# B&R Automation Studio project BaseProject (part 6)

#### Main.st
```iecst
(*******************************************************************************
 * Copyright: B&R Industrial Automation
 * Author:    Tyler Matijevich
 * Created:   November 5, 2020/12:35
********************************************************************************
 * Description: Control program to handle assembly power commands and error
 statuses
********************************************************************************)

PROGRAM _INIT

END_PROGRAM

PROGRAM _CYCLIC

	fbTrakModule(MpLink := ADR(TrackInterface.ModulePml),
					Enable := TRUE,
					Parameters := ADR(parTrakModule));

	// Reset command if no error
	IF gTrakSystem.Asm.Status.Error = FALSE THEN
		gTrakSystem.Asm.Cmd.ErrorReset := FALSE; // Force this command to reset
	END_IF

	(****************************************************************************************************
	****************************************************************************************************)
	(*
		Interrupts:
		1. Error status
		2. Stop command
		3. Read error
		4. ErrorStop state
	*)

	// 1. Skip remaining interrupt checks when an error exists
	IF gTrakSystem.Asm.Status.Error OR ShInit.Status.Error THEN
		// Go to ERROR
		AssemblyState := ASM_STATE_ERROR;

	// 2. Accept stop command
	ELSIF gTrakSystem.Asm.Cmd.Stop THEN
		// Power off if powering or powered on
		IF gTrakSystem.Asm.Status.Homing OR gTrakSystem.Asm.Status.Ready THEN
			// Execute the power off command. Execute should not be true in either of these states
			fbAsmPowerOff.Execute := TRUE;
		END_IF

		// Go to OFF
		AssemblyState := ASM_STATE_OFF;

	// 3. The assembly read function blocks are in error
	ELSIF fbAsmReadStatus.Error OR fbAsmReadInfo.Error THEN
		// Log event
		// Set error status and go to ERROR
		gTrakSystem.Asm.Status.Error	:= TRUE;
		AssemblyState 				:= ASM_STATE_ERROR;

	// 4. Assembly in ErrorStop
	ELSIF gTrakSystem.Asm.Status.ErrorStop AND fbAsmReset.Busy = FALSE THEN
		// Log event
		// Set error status and go to ERROR
		gTrakSystem.Asm.Status.Error	:= TRUE;
		AssemblyState 				:= ASM_STATE_ERROR;

	END_IF

	(****************************************************************************************************
	****************************************************************************************************)
	// Main assembly state machine
	CASE AssemblyState OF
		// ----------------------------------------------------------------------------------------------------
		// OFF
		ASM_STATE_OFF:
			// Accept AsmPowerOff command
			IF fbAsmPowerOff.Done THEN
				// Reset execution
				fbAsmPowerOff.Execute := FALSE;

			ELSIF fbAsmPowerOff.Error THEN
				// Log event
				// Set error status and go to ERROR
				gTrakSystem.Asm.Status.Error	:= TRUE;
				AssemblyState 				:= ASM_STATE_ERROR;

			// Accept AsmReset command
			ELSIF fbAsmReset.Done THEN
				// Reset execution
				fbAsmReset.Execute := FALSE;

			ELSIF fbAsmReset.Error THEN
				// Log event
				// Set error status and go to ERROR
				gTrakSystem.Asm.Status.Error	:= TRUE;
				AssemblyState 				:= ASM_STATE_ERROR;

			// Wait for power command and assembly conditions
			ELSIF gTrakSystem.Asm.Cmd.Power AND gTrakSystem.Asm.Cmd.Stop = FALSE // Read input commands
			  AND gTrakSystem.Asm.Status.Disabled AND gTrakSystem.Asm.Status.ReadyForPowerOn // Check assembly statuses
			  AND fbAsmPowerOff.Execute = FALSE AND fbAsmReset.Execute = FALSE
			  AND MpPackMLStateIsActive(TrackInterface.ModulePml,mpPACKML_STATE_EXECUTE,1)
			  	THEN // Check other function block execution
				// Power on the assembly
				fbAsmPowerOn.Execute := TRUE;

				// Go to POWER
				AssemblyState := ASM_STATE_POWER;

			END_IF

		// ----------------------------------------------------------------------------------------------------
		// POWER
		ASM_STATE_POWER:
			// Wait for the power on command to complete, ensure correct statuses
			IF fbAsmPowerOn.Done AND gTrakSystem.Asm.Status.Ready AND gTrakSystem.Asm.Status.PowerOn THEN
				// Reset execution
				fbAsmPowerOn.Execute := FALSE;

				// Go to READY
				AssemblyState := ASM_STATE_READY;

//				// Check shuttle initialization for ready status
//				IF ShInit.Status.Ready THEN
//					// Start the shuttle initialization
//					ShInit.Cmd.Start := TRUE;
//
//					// Go to INIT
//					AssemblyState := ASM_STATE_INIT;
//
//				ELSE
//					// Log event
//					// Set error status and go to ERROR
//					gTrakSystem.Asm.Status.Error	:= TRUE;
//					AssemblyState 				:= ASM_STATE_ERROR;
//
//				END_IF

			ELSIF fbAsmPowerOn.Error THEN
				// Log event
				// Set error status and go to ERROR
				gTrakSystem.Asm.Status.Error	:= TRUE;
				AssemblyState 				:= ASM_STATE_ERROR;

			// Check if the assembly suddenly loses power
			ELSIF (gTrakSystem.Asm.Status.Disabled OR gTrakSystem.Asm.Status.PowerOn = FALSE)
			  AND fbAsmPowerOn.Execute = FALSE THEN
				// Log event
				// Set error status and go to ERROR
				gTrakSystem.Asm.Status.Error	:= TRUE;
				AssemblyState 				:= ASM_STATE_ERROR;

			END_IF

		// ----------------------------------------------------------------------------------------------------
		// INIT
		ASM_STATE_INIT:
		// Go to READY
				AssemblyState := ASM_STATE_READY;

			// Wait for the shuttle initialization to complete
//			IF ShInit.Status.Complete THEN
//				// Reset command
//				ShInit.Cmd.Start := FALSE;
//
//				// Go to READY
//				AssemblyState := ASM_STATE_READY;
//
//			ELSIF ShInit.Status.Error THEN
//				// Log event
//				// Set error status and go to ERROR
//				gTrakSystem.Asm.Status.Error	:= TRUE;
//				AssemblyState 				:= ASM_STATE_ERROR;
//
//			END_IF

		// ----------------------------------------------------------------------------------------------------
		// READY
		ASM_STATE_READY:
			// Check if the assembly suddenly becomes disabled
			IF gTrakSystem.Asm.Status.Disabled THEN
				// Log event
				// Set error status and go to ERROR
				gTrakSystem.Asm.Status.Error	:= TRUE;
				AssemblyState 				:= ASM_STATE_ERROR;

			END_IF

		// ----------------------------------------------------------------------------------------------------
		// ERROR
		ASM_STATE_ERROR:
			// Wait for an error reset command
			IF gTrakSystem.Asm.Cmd.ErrorReset THEN
				// If ErrorStop, reset the assembly
				IF gTrakSystem.Asm.Status.ErrorStop AND fbAsmReset.Error = FALSE THEN
					// Execute an assembly reset
					fbAsmReset.Execute := TRUE;

					// Reset other function block's execution
					fbAsmPowerOn.Execute 	:= FALSE;
					fbAsmPowerOff.Execute	:= FALSE;

				// If powered
				ELSIF (gTrakSystem.Asm.Status.Homing OR gTrakSystem.Asm.Status.Ready) AND fbAsmPowerOff.Error = FALSE THEN
					// Power off the assembly
					fbAsmPowerOff.Execute := TRUE;

					// Reset other function block's execution
					fbAsmPowerOn.Execute 	:= FALSE;
					fbAsmReset.Execute		:= FALSE;

				ELSE
					// Reset all function block's execution
					fbAsmPowerOn.Execute 	:= FALSE;
					fbAsmPowerOff.Execute	:= FALSE;
					fbAsmReset.Execute		:= FALSE;

				END_IF // Check assembly state

				// Reset the error bit and go back to OFF
				gTrakSystem.Asm.Status.Error	:= FALSE;
				AssemblyState				:= ASM_STATE_OFF;

			END_IF

	END_CASE // Assembly state machine

	// Call all mapp Trak function blocks
	fbAsmReadStatus(Assembly := ADR(TrackInterface.SampleTrak), Enable := TRUE); // Always enable to reduce logger entries
	fbAsmReadInfo(Assembly := ADR(TrackInterface.SampleTrak), Enable := TRUE); // Always enable to reduce logger entries
	fbAsmPowerOn(Assembly := ADR(TrackInterface.SampleTrak));
	fbAsmPowerOff(Assembly := ADR(TrackInterface.SampleTrak));
	fbAsmReset(Assembly := ADR(TrackInterface.SampleTrak));

	// Update the global status information
	gTrakSystem.Asm.Status.Disabled					:= fbAsmReadStatus.Valid AND fbAsmReadStatus.AssemblyDisabled;
	gTrakSystem.Asm.Status.Homing					:= fbAsmReadStatus.Valid AND fbAsmReadStatus.AssemblyHoming;
	gTrakSystem.Asm.Status.Ready					:= fbAsmReadStatus.Valid AND fbAsmReadStatus.AssemblyReady;
	gTrakSystem.Asm.Status.Stopping					:= fbAsmReadStatus.Valid AND fbAsmReadStatus.AssemblyStopping;
	gTrakSystem.Asm.Status.ErrorStop				:= fbAsmReadStatus.Valid AND fbAsmReadStatus.AssemblyErrorStop;
	gTrakSystem.Asm.Status.CommunicationReady		:= fbAsmReadInfo.Valid AND fbAsmReadInfo.AssemblyInfo.CommunicationReady;
	gTrakSystem.Asm.Status.ReadyForPowerOn			:= fbAsmReadInfo.Valid AND fbAsmReadInfo.AssemblyInfo.ReadyForPowerOn;
	gTrakSystem.Asm.Status.PowerOn					:= fbAsmReadInfo.Valid AND fbAsmReadInfo.AssemblyInfo.PowerOn;
	gTrakSystem.Asm.Status.ShuttlesInErrorStopCount	:= fbAsmReadInfo.AssemblyInfo.ShuttlesInErrorStopCount; // If not valid, assuming these are zero
	gTrakSystem.Asm.Status.StartupCount				:= fbAsmReadInfo.AssemblyInfo.StartupCount;

	// Call all subroutine actions
	ShInit.Cmd.Stop := gTrakSystem.Asm.Status.Ready = FALSE;
//	ShuttleInitialization;

END_PROGRAM

PROGRAM _EXIT

END_PROGRAM
```

### SM11.var
```iecst
(*Shuttle initialization variables*)
VAR
	BufferReturnIndex : TrBaseErrorCodeEnum;
	fbAsmGetShuttle : MC_BR_AsmGetShuttle_AcpTrak;
	fbShCopyUserData : MC_BR_ShCopyUserData_AcpTrak;
END_VAR
```

### Program Logical/Source/SampleTrak/Assembly/SubModule1/ShuttleInit (IEC)

#### Main.st
```iecst
PROGRAM _INIT
	(* Insert code here *)
	 TrakInterface;
END_PROGRAM

PROGRAM _CYCLIC
	// Reset status variables, they will be set in the respective state
	ShInit.Status.Ready 	:= FALSE;
	ShInit.Status.Complete	:= FALSE;

	(*
		Interrupts:
		1. Error status
		2. Stop command
	*)
	// 1. Check error status
	IF ShInit.Status.Error THEN
		// Go to ERROR, skip remaining interrupts
		ShInitState := 255;

	// 2. Accept stop commands
	ELSIF ShInit.Cmd.Stop THEN
		// Reset FB execution
		fbAsmGetShuttle.Enable		:= FALSE;
		fbShCopyUserData.Execute 	:= FALSE;

		// Go to INIT
		ShInitState := 0;

	END_IF

	// Shuttle initialization main state machine
	CASE ShInitState OF
		// ----------------------------------------------------------------------------------------------------
		// INIT
		0:
			// Set the status
			ShInit.Status.Ready := TRUE;

			// Wait to start
			IF ShInit.Cmd.Start AND ShInit.Cmd.Stop = FALSE THEN
				// Clear the shuttle buffer
				BufferReturnIndex := TrBaseClearShBuffer(ADR(gTrakSystem.Buffer), SIZEOF(gTrakSystem.Buffer));
				IF BufferReturnIndex = trBASE_NO_ERROR THEN
					// Enable the assembly get shuttle function block
					fbAsmGetShuttle.Assembly 	:= ADR(TrakInterface.SampleTrak);
					fbAsmGetShuttle.Enable 		:= TRUE;

					// Go to READ
					ShInitState := 10;

				ELSE
					// Log event
					// Set error status and go to ERROR
					ShInit.Status.Error := TRUE;
					ShInitState 		:= 255;

				END_IF
			END_IF // Start

		// ----------------------------------------------------------------------------------------------------
		// READ
		10:
			// Wait for a valid read, then read the shuttle
			IF fbAsmGetShuttle.Valid AND fbAsmGetShuttle.TotalCount > 0 THEN
				// Add the shuttle to the buffer
				BufferReturnIndex := TrBaseAddShToBuffer(fbAsmGetShuttle.Axis, ADR(gTrakSystem.Buffer), SIZEOF(gTrakSystem.Buffer));
				IF BufferReturnIndex = trBASE_NO_ERROR THEN
					// Shuttle added successfully, read the shuttle user data
					fbShCopyUserData.Axis 			:= ADR(fbAsmGetShuttle.Axis);
					fbShCopyUserData.DataAddress	:= ADR(ShuttleUserData);
					fbShCopyUserData.DataSize		:= SIZEOF(ShuttleUserData);
					fbShCopyUserData.Mode			:= mcACPTRAK_USERDATA_GET;
					fbShCopyUserData.Execute		:= TRUE;

					// Go to DATA
					ShInitState := 20;

				ELSE
					// Log event
					// Set error status and go to ERROR
					ShInit.Status.Error := TRUE;
					ShInitState 		:= 255;

				END_IF

			ELSIF fbAsmGetShuttle.Valid AND fbAsmGetShuttle.TotalCount = 0 THEN // No shuttles on the assembly
				// Go straight to the complete state
				ShInitState := 60;

			ELSIF fbAsmGetShuttle.Error THEN
				// Log event
				// Set error status and go to ERROR
				ShInit.Status.Error := TRUE;
				ShInitState 		:= 255;

			END_IF

		// ----------------------------------------------------------------------------------------------------
		// DATA
		20:
			IF fbShCopyUserData.Done THEN
				// Reset the command
				fbShCopyUserData.Execute := FALSE;

				// Go to WRITE
				ShInitState := 30;

			ELSIF fbShCopyUserData.Error THEN
				// Log event
				// Set error status and go to ERROR
				ShInit.Status.Error := TRUE;
				ShInitState 		:= 255;

			END_IF

		// ----------------------------------------------------------------------------------------------------
		// WRITE
		30:
			IF fbShCopyUserData.Done THEN
				// Shuttle user data write complete, shuttle ID set, reset the execution
				fbShCopyUserData.Execute := FALSE;

				// Reset the assembly get shuttle next command
				fbAsmGetShuttle.Next := FALSE;

				// Go to UPDATE
				ShInitState := 40;

			ELSIF fbShCopyUserData.Error THEN
				// Log event
				// Set error status and go to ERROR
				ShInit.Status.Error := TRUE;
				ShInitState 		:= 255;

			ELSE
				// Execute the write command
				fbShCopyUserData.Mode		:= mcACPTRAK_USERDATA_SET;
				fbShCopyUserData.Execute 	:= TRUE;

				// Set the shuttle ID (if not already set)
				ShuttleUserData.ID := fbAsmGetShuttle.AdditionalInfo.ShuttleID;

			END_IF

		// ----------------------------------------------------------------------------------------------------
		// UPDATE
		40:
			// Check for the next shuttle
			IF fbAsmGetShuttle.Valid AND fbAsmGetShuttle.RemainingCount > 0 THEN
				// Issue next command and go back to the READ state
				fbAsmGetShuttle.Next 	:= TRUE;
				ShInitState				:= 10;

			// Check when no shuttles remain
			ELSIF fbAsmGetShuttle.Valid AND fbAsmGetShuttle.RemainingCount = 0 THEN
				// All shuttles have been captured, reset the FB
				fbAsmGetShuttle.Enable := FALSE;

				// Go to DELETE
				ShInitState := 50;

			ELSIF fbAsmGetShuttle.Error THEN
				// Log event
				// Set error status and go to ERROR
				ShInit.Status.Error := TRUE;
				ShInitState 		:= 255;

			END_IF

		// ----------------------------------------------------------------------------------------------------
		// DELETE
		50:
			// Shuttle detection complete, now delete marked shuttles
			gTrakSystem.Tracking.Cmd.Delete := gTrakSystem.Tracking.Status.ShuttlesToBeDeletedCount <> 0;

			// Leave when no shuttles need to be deleted
			IF gTrakSystem.Tracking.Status.ShuttlesToBeDeletedCount = 0 THEN
				// Go to COMPLETE
				ShInitState := 60;
			END_IF

		// ----------------------------------------------------------------------------------------------------
		// COMPLETE
		60:
			// Set the status
			ShInit.Status.Complete := TRUE;

			// Return to INIT when the state command is reset
			IF ShInit.Cmd.Start = FALSE THEN
				// Go to INIT
				ShInitState := 0;
			END_IF

		// ----------------------------------------------------------------------------------------------------
		// ERROR
		255:
			// Wait for error reset command
			IF ShInit.Cmd.ErrorReset THEN
				// Reset the function blocks
				fbAsmGetShuttle.Enable 		:= FALSE;
				fbShCopyUserData.Execute 	:= FALSE;

				// Reset the error bit and go to INIT
				ShInit.Status.Error := FALSE;
				ShInitState 		:= 0;

			END_IF

	END_CASE

	// Call mapp Trak function blocks
	fbAsmGetShuttle();
	fbShCopyUserData();

END_PROGRAM

PROGRAM _EXIT
	(* Insert code here *)

END_PROGRAM
```

### Program Logical/Source/SampleTrak/Assembly/Alarm

#### Variables.var
```iecst
VAR
	fbAlarmTrakModule : MpAlarmXCore;
	FilterConfiguration : STRING[1000] := '';
	SortConfiguration : STRING[1000] := '';
	HistoryFilter : STRING[2000] := '';
	HistorySort : STRING[2000] := '';
	TriggerTestAlarm : BOOL;
END_VAR
```

#### Main.st
```iecst
PROGRAM _INIT
	(* Insert code here *)
	FilterConfiguration;
	SortConfiguration;
	HistoryFilter;
	HistorySort;

END_PROGRAM

PROGRAM _CYCLIC
	(* Insert code here *)

	fbAlarmTrakModule(MpLink := ADR(gAlarmXCore_TrakModule), Enable := TRUE);

	TriggerTestAlarm;

END_PROGRAM

PROGRAM _EXIT
	(* Insert code here *)

END_PROGRAM
```

### Package Logical/Source/SampleTrak/ReusableSource - EquipmentModuleSource

### Source.var
```iecst
VAR
	ModuleLink : STRING[40];
	ModuleName : STRING[40];
	StartValue : INT;
	Counter : INT;
	StartValu : INT;
	ModuleInterface : ModuleInterfaceType;
END_VAR
(*Alarm configuration*)
VAR
	fbAlarmModule : MpAlarmXCore;
	FilterConfiguration : STRING[1000] := '';
	SortConfiguration : STRING[1000] := '';
	HistoryFilter : STRING[2000] := '';
	HistorySort : STRING[2000] := '';
	ConfigAlarm : BOOL;
	ConfigWarning : BOOL;
	ConfigInformation : BOOL;
	RecoveryAlarm : BOOL;
	RecoveryWarning : BOOL;
	RecoveryInformation : BOOL;
	OperationAlarm : BOOL;
	OperationWarning : BOOL;
	OperationInformation : BOOL;
	fbModuleConfig : MpRecipeXml;
	ConfigCategory : STRING[50];
	ConfigHeader : MpRecipeXmlHeaderType;
	fbConfigRegPar : MpRecipeRegPar;
END_VAR
```

### Source.typ
```iecst
TYPE
	ModuleInterfaceType : 	STRUCT
		SampleTrak : McAssemblyType;
		MainPml : MpComIdentType;
		ModulePml : MpComIdentType;
		AlarmCore : MpComIdentType;
	END_STRUCT;
END_TYPE
```

### Program Logical/Source/SampleTrak/ReusableSource/Config (IEC)

#### Main.st
```iecst
PROGRAM _INIT
	(* Read out the task name for multiple deployed programs for in line configuration *)

	ST_name(0,ADR(ModuleLink),0);

	IF (ModuleLink = 'EM2::Config2') THEN

		ModuleName := 'EM2';
		ConfigCategory := ModuleName;
		ConfigHeader.Version := '0.0.1';
		StartValue := 0;

	ELSIF (ModuleLink = 'EM3::Config3') THEN

		ModuleName := 'EM3';
		ConfigCategory := ModuleName;
		ConfigHeader.Version := '0.0.1';
		StartValue := 10000;

	END_IF

	Counter := StartValue;

	//call each AppModule based MpLinks so it variable exists in memory and can be used in the AppModule variable mapping
	gRecipeXml_EM2;
	gRecipeXml_EM3;
	gPackMLModule_EM2;
	gPackMLModule_EM3;

END_PROGRAM

PROGRAM _CYCLIC
	(* Insert code here *)
	ConfigAlarm;
	ConfigWarning;
	ConfigInformation;

	fbModuleConfig(MpLink := ADR(ModuleInterface.RecipeCore),
			Enable := TRUE,
			DeviceName := ADR('Config'),
			FileName := ADR(ModuleName),
			Header := ADR(ConfigHeader),
			Category := ADR(ConfigCategory));

	fbConfigRegPar(MpLink := ADR(ModuleInterface.RecipeCore), Enable := TRUE , PVName := ADR('ModuleInterface'), Category := ADR(ConfigCategory));

END_PROGRAM

PROGRAM _EXIT
	(* Insert code here *)

END_PROGRAM
```

### Program Logical/Source/SampleTrak/ReusableSource/Operation (IEC)

#### Main.st
```iecst
PROGRAM _INIT
	(* Insert code here *)

END_PROGRAM

PROGRAM _CYCLIC
	(* This is just a test *)

	IF MpPackMLStateIsActive(ModuleInterface.MainPml,mpPACKML_STATE_EXECUTE,1) THEN
		Counter := Counter + 1;
	END_IF

	OperationAlarm;
	OperationWarning;
	OperationInformation;

END_PROGRAM

PROGRAM _EXIT
	(* Insert code here *)

END_PROGRAM
```

### Program Logical/Source/SampleTrak/ReusableSource/Recovery (IEC)

#### Main.st
```iecst
PROGRAM _INIT
	(* Insert code here *)

END_PROGRAM

PROGRAM _CYCLIC
	(* Insert code here *)
	RecoveryAlarm;
	RecoveryWarning;
	RecoveryInformation;

END_PROGRAM

PROGRAM _EXIT
	(* Insert code here *)

END_PROGRAM
```

### Package Logical/Source/SampleTrak/EMx - EquipmentModule2

### EMx.var
```iecst
VAR
	ModuleInterface : ModuleInterfaceType;
END_VAR
```

### Program Logical/Source/SampleTrak/EMx/Process (IEC)

#### Variables.var
```iecst
VAR
	MpAlarmX : MpComIdentType;
	ModuleName : STRING[30];
	StartValue : INT;
	Counter : INT;
	MpLink : REFERENCE TO MpComIdentType;
END_VAR
```

#### Main.st
```iecst
PROGRAM _INIT
	(* Insert code here *)

	ST_name(0,ADR(ModuleName),0);

	IF (ModuleName = 'EM12::Process1') THEN

		StartValue := 1000;

	ELSIF (ModuleName = 'EM12::Process2') THEN

		StartValue := 0;

	ELSIF (ModuleName = 'EM12::Process3') THEN

		StartValue := 15000;

	END_IF

	Counter := StartValue;

	MpAlarmX;

END_PROGRAM

PROGRAM _CYCLIC
	(* Insert code here *)
	IF MpPackMLStateIsActive(ModuleInterface.MainPml,mpPACKML_STATE_EXECUTE,1) THEN
		Counter := Counter + 1;
	END_IF

END_PROGRAM

PROGRAM _EXIT
	(* Insert code here *)

END_PROGRAM
```

### Program Logical/Source/SampleTrak/Main

#### Main.st
```iecst
PROGRAM _INIT
	(* Call version control variables so they can be updated during every project build *)
	 MachineLastRevisionDate;
	 MachineSoftwareVersion;

END_PROGRAM

PROGRAM _CYCLIC
	(*  Insert code here *)

END_PROGRAM

PROGRAM _EXIT
	(* Insert code here *)

END_PROGRAM
```

- gSampleTrak.wsp (not shown)

- Visualisation Logical/mappView (not shown)

- Project.language (not shown)

### MachineVersionInfo.var - not listed in the package file held
```iecst
VAR
	MachineSoftwareVersion : STRING[80] := 'dev-FWimporter-1.2.0-80-23721ca';
	MachineLastRevisionDate : DATE_AND_TIME := DT#2022-07-21-11:17;
END_VAR
```

Listed in the project but not available here: Logical/Libraries/TrBase/TrBase.var, Logical/Libraries/TrkDiag/TrkDiag.var, Logical/Source/Diagnostic/TrakDiagGlobal.typ, Logical/Source/Diagnostic/DiagConfig/Cyclic.st, Logical/Source/Diagnostic/TrackDiag/Exit.st, Logical/Source/EMx/EMx.typ, Logical/Source/ReusableSource/Source.typ, Logical/Source/ReusableSource/Config, Logical/Source/ReusableSource/Operation, Logical/Source/ReusableSource/Recovery, Logical/Source/SampleTrak/SampleTrak.var, Logical/Source/SampleTrak/TSMMain/Types.typ, Logical/Source/SampleTrak/TSMMain/Variables.var, Logical/Source/SampleTrak/TSMMain/Main.st, Logical/Source/SampleTrak/Diagnostic/DiagConfig/Cyclic.st, Logical/Source/SampleTrak/Diagnostic/DiagConfig/Exit.st, Logical/Source/SampleTrak/Diagnostic/DiagConfig/Types.typ, Logical/Source/SampleTrak/Diagnostic/DiagConfig/Variables.var, Logical/Source/SampleTrak/Assembly/SubModule1/SM11.typ, Logical/Source/SampleTrak/ReusableSource/BarrierCtrl, Logical/Source/SampleTrak/ReusableSource/Alarm, Logical/Source/SampleTrak/EMx/EMx.typ, Logical/UserData/SegTrace
